KUKA KRL program: edge_4_right_mte.src, edge_4_right_mte.dat

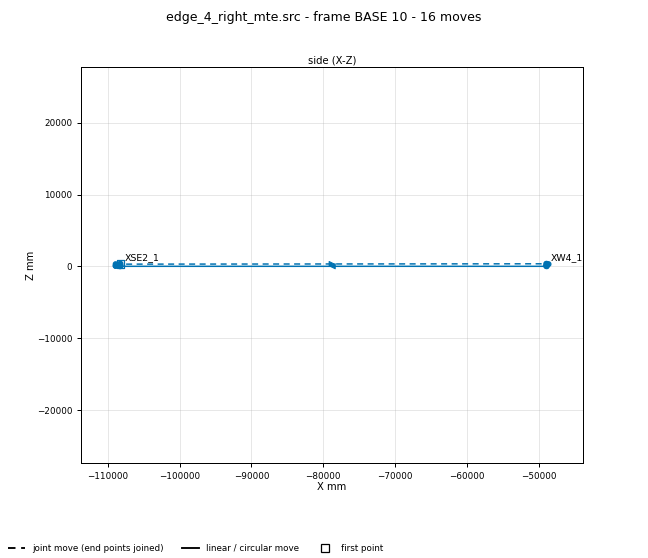
[picture p0: tool path of edge_4_right_mte.src in frame BASE 10, 16 of 16 moves have a stored position in this frame; points joined in program order, loops and branches not executed]
--- edge_4_right_mte.src ---
&ACCESS RVP
&REL 45
&PARAM EDITMASK = *
&PARAM DISKPATH = KRC:\R1\Program
DEF edge_4_right_mte( )
;FOLD INI;%{PE}
  ;FOLD BASISTECH INI
    GLOBAL INTERRUPT DECL 3 WHEN $STOPMESS==TRUE DO IR_STOPM ( )
    INTERRUPT ON 3
    BAS (#INITMOV,0 )
  ;ENDFOLD (BASISTECH INI)
  ;FOLD USER INI
    ;Make your modifications here

  ;ENDFOLD (USER INI)
;ENDFOLD (INI)
TS_CorrOff()
;FOLD PTP SE2_1 Vel= 100 % PDATW1_1 Tool[1] Base[10] ;%{PE}%R 8.3.34,%MKUKATPBASIS,%CMOVE,%VPTP,%P 1:PTP, 2:SE2_1, 3:C_DIS, 5:100, 7:PDATSE2_1
$BWDSTART = FALSE
PDAT_ACT=PPDATSE2_1
FDAT_ACT=FSE2_1
BAS(#PTP_PARAMS,100)
SET_CD_PARAMS (0)
PTP XSE2_1 C_DIS
;ENDFOLD

;FOLD LIN SE2_2 Vel= 0.06 m/s CPDATSE2_2 TouchSense SEARCH VIA SE2_3 CDSE2_2 SPSE2_2 Tool[1] Base[10] ;%{PE}
;FOLD Parameters ;%{h}
;Params IlfProvider=kukaroboter.touchsense.searchlin; Kuka.PointName=SE2_2; Kuka.BlendingEnabled=False; Kuka.MoveDataName=CPDATSE2_2; Kuka.VelocityPath=0.06; Kuka.MovementParameterFieldEnabled=True; MoveType=LIN
;FOLD Parameters TouchSense ;%{h}
;Params TouchSense.SearchViaPoint=SE2_3;TouchSense.ReferenceMove=CDSE2_2;TouchSense.SeachParam=SPSE2_2
;ENDFOLD
;ENDFOLD
$BWDSTART = FALSE
LDAT_ACT=LCPDATSE2_2
FDAT_ACT=FSE2_2
BAS(#CP_PARAMS,0.06)
SET_CD_PARAMS (0)
LIN XSE2_2 C_DIS C_DIS
TS_InitMovement($POS_ACT, XSE2_3, ZSPSE2_2)
TS_ManMoveToVia(XSE2_3)
TS_Search(XSE2_3, ZSPSE2_2, VCDSE2_2)
TS_SetCorrData(ZSPSE2_2, VCDSE2_2)
;ENDFOLD

;FOLD TouchSense Corr 1 CDSE2_2;%{E}
;FOLD Parameters Corr 1D ;%{h}
;Params IlfProvider=KukaRoboter.TouchSense.Correction1D;Correction1D=CDSE2_2
;ENDFOLD
TS_BC6DCalc(VCDSE2_2, TSg_CD0, TSg_CD0, TSg_CD0, TSg_CD0, TSg_CD0)
;ENDFOLD

;FOLD LIN SE2_4 Vel= 0.06 m/s CPDATSE2_4 TouchSense SEARCH VIA SE2_5 CDSE2_4 SPSE2_4 Tool[1] Base[10] ;%{PE}
;FOLD Parameters ;%{h}
;Params IlfProvider=kukaroboter.touchsense.searchlin; Kuka.PointName=SE2_4; Kuka.BlendingEnabled=False; Kuka.MoveDataName=CPDATSE2_4; Kuka.VelocityPath=0.06; Kuka.MovementParameterFieldEnabled=True; MoveType=LIN
;FOLD Parameters TouchSense ;%{h}
;Params TouchSense.SearchViaPoint=SE2_5;TouchSense.ReferenceMove=CDSE2_4;TouchSense.SeachParam=SPSE2_4
;ENDFOLD
;ENDFOLD
$BWDSTART = FALSE
LDAT_ACT=LCPDATSE2_4
FDAT_ACT=FSE2_4
BAS(#CP_PARAMS,0.06)
SET_CD_PARAMS (0)
LIN XSE2_4 C_DIS C_DIS
TS_InitMovement($POS_ACT, XSE2_5, ZSPSE2_4)
TS_ManMoveToVia(XSE2_5)
TS_Search(XSE2_5, ZSPSE2_4, VCDSE2_4)
TS_SetCorrData(ZSPSE2_4, VCDSE2_4)
;ENDFOLD

;FOLD TouchSense Corr 2 CDSE2_2 CDSE2_4;%{E}
;FOLD Parameters Corr 2D ;%{h}
;Params IlfProvider=KukaRoboter.TouchSense.Correction2D;Correction1D=CDSE2_2;Correction2D=CDSE2_4
;ENDFOLD
TS_BC6DCalc(VCDSE2_2, TSg_CD0, TSg_CD0, VCDSE2_4, TSg_CD0, TSg_CD0)
;ENDFOLD

;FOLD LIN SE2_6 Vel= 0.06 m/s CPDATS1_2 Tool[1] Base[10] ;%{PE}%R 8.3.34,%MKUKATPBASIS,%CMOVE,%VLIN,%P 1:LIN, 2:SE2_6, 3:, 5:0.06, 7:CPDATSE2_6
$BWDSTART = FALSE
LDAT_ACT=LCPDATSE2_6
FDAT_ACT=FSE2_6
BAS(#CP_PARAMS,0.06)
SET_CD_PARAMS (0)
LIN XSE2_6 C_DIS C_DIS
;ENDFOLD

;FOLD LIN SE2_7 Vel= 0.02 m/s CPDATSE2_7 TouchSense SEARCH VIA SE2_8 CDSE2_7 SPSE2_7 Tool[1] Base[10] ;%{PE}
;FOLD Parameters ;%{h}
;Params IlfProvider=kukaroboter.touchsense.searchlin; Kuka.PointName=SE2_7; Kuka.BlendingEnabled=False; Kuka.MoveDataName=CPDATSE2_7; Kuka.VelocityPath=0.02; Kuka.MovementParameterFieldEnabled=True; MoveType=LIN
;FOLD Parameters TouchSense ;%{h}
;Params TouchSense.SearchViaPoint=SE2_8;TouchSense.ReferenceMove=CDSE2_7;TouchSense.SeachParam=SPSE2_7
;ENDFOLD
;ENDFOLD
$BWDSTART = FALSE
LDAT_ACT=LCPDATSE2_7
FDAT_ACT=FSE2_7
BAS(#CP_PARAMS,0.02)
SET_CD_PARAMS (0)
LIN XSE2_7 C_DIS C_DIS
TS_InitMovement($POS_ACT, XSE2_8, ZSPSE2_7)
TS_ManMoveToVia(XSE2_8)
TS_Search(XSE2_8, ZSPSE2_7, VCDSE2_7)
TS_SetCorrData(ZSPSE2_7, VCDSE2_7)
;ENDFOLD

;FOLD TouchSense Corr 3 CDSE2_2 CDSE2_4 CDSE2_7;%{E}
;FOLD Parameters Corr 3D ;%{h}
;Params IlfProvider=KukaRoboter.TouchSense.Correction3D;Correction1D=CDSE2_2;Correction2D=CDSE2_4;Correction3D=CDSE2_7
;ENDFOLD
TS_BC6DCalc(VCDSE2_2, TSg_CD0, TSg_CD0, VCDSE2_4, TSg_CD0, VCDSE2_7)
;ENDFOLD

;FOLD LIN SE2_9 Vel= 0.1 m/s CPDATS1_2 Tool[1] Base[10] ;%{PE}%R 8.3.34,%MKUKATPBASIS,%CMOVE,%VLIN,%P 1:LIN, 2:SE2_9, 3:, 5:0.1, 7:CPDATSE2_9
$BWDSTART = FALSE
LDAT_ACT=LCPDATSE2_9
FDAT_ACT=FSE2_9
BAS(#CP_PARAMS,0.1)
SET_CD_PARAMS (0)
LIN XSE2_9 C_DIS C_DIS
;ENDFOLD

;FOLD PTP SS3_1 Vel= 100 % PDATW1_1 Tool[1] Base[10] ;%{PE}%R 8.3.34,%MKUKATPBASIS,%CMOVE,%VPTP,%P 1:PTP, 2:SS3_1, 3:C_DIS, 5:100, 7:PDATSS3_1
$BWDSTART = FALSE
PDAT_ACT=PPDATSS3_1
FDAT_ACT=FSS3_1
BAS(#PTP_PARAMS,100)
SET_CD_PARAMS (0)
PTP XSS3_1 C_DIS
;ENDFOLD

;FOLD LIN SS3_2 Vel= 0.06 m/s CPDATSS3_2 TouchSense SEARCH VIA SS3_3 CDSS3_2 SPSS3_2 Tool[1] Base[10] ;%{PE}
;FOLD Parameters ;%{h}
;Params IlfProvider=kukaroboter.touchsense.searchlin; Kuka.PointName=SS3_2; Kuka.BlendingEnabled=False; Kuka.MoveDataName=CPDATSS3_2; Kuka.VelocityPath=0.06; Kuka.MovementParameterFieldEnabled=True; MoveType=LIN
;FOLD Parameters TouchSense ;%{h}
;Params TouchSense.SearchViaPoint=SS3_3;TouchSense.ReferenceMove=CDSS3_2;TouchSense.SeachParam=SPSS3_2
;ENDFOLD
;ENDFOLD
$BWDSTART = FALSE
LDAT_ACT=LCPDATSS3_2
FDAT_ACT=FSS3_2
BAS(#CP_PARAMS,0.06)
SET_CD_PARAMS (0)
LIN XSS3_2 C_DIS C_DIS
TS_InitMovement($POS_ACT, XSS3_3, ZSPSS3_2)
TS_ManMoveToVia(XSS3_3)
TS_Search(XSS3_3, ZSPSS3_2, VCDSS3_2)
TS_SetCorrData(ZSPSS3_2, VCDSS3_2)
;ENDFOLD

;FOLD TouchSense Corr 1 CDSS3_2;%{E}
;FOLD Parameters Corr 1D ;%{h}
;Params IlfProvider=KukaRoboter.TouchSense.Correction1D;Correction1D=CDSS3_2
;ENDFOLD
TS_BC6DCalc(VCDSS3_2, TSg_CD0, TSg_CD0, TSg_CD0, TSg_CD0, TSg_CD0)
;ENDFOLD

;FOLD LIN SS3_4 Vel= 0.06 m/s CPDATSS3_4 TouchSense SEARCH VIA SS3_5 CDSS3_4 SPSS3_4 Tool[1] Base[10] ;%{PE}
;FOLD Parameters ;%{h}
;Params IlfProvider=kukaroboter.touchsense.searchlin; Kuka.PointName=SS3_4; Kuka.BlendingEnabled=False; Kuka.MoveDataName=CPDATSS3_4; Kuka.VelocityPath=0.06; Kuka.MovementParameterFieldEnabled=True; MoveType=LIN
;FOLD Parameters TouchSense ;%{h}
;Params TouchSense.SearchViaPoint=SS3_5;TouchSense.ReferenceMove=CDSS3_4;TouchSense.SeachParam=SPSS3_4
;ENDFOLD
;ENDFOLD
$BWDSTART = FALSE
LDAT_ACT=LCPDATSS3_4
FDAT_ACT=FSS3_4
BAS(#CP_PARAMS,0.06)
SET_CD_PARAMS (0)
LIN XSS3_4 C_DIS C_DIS
TS_InitMovement($POS_ACT, XSS3_5, ZSPSS3_4)
TS_ManMoveToVia(XSS3_5)
TS_Search(XSS3_5, ZSPSS3_4, VCDSS3_4)
TS_SetCorrData(ZSPSS3_4, VCDSS3_4)
;ENDFOLD

;FOLD TouchSense Corr 2 CDSS3_2 CDSS3_4;%{E}
;FOLD Parameters Corr 2D ;%{h}
;Params IlfProvider=KukaRoboter.TouchSense.Correction2D;Correction1D=CDSS3_2;Correction2D=CDSS3_4
;ENDFOLD
TS_BC6DCalc(VCDSS3_2, TSg_CD0, TSg_CD0, VCDSS3_4, TSg_CD0, TSg_CD0)
;ENDFOLD

;FOLD LIN SS3_6 Vel= 0.1 m/s CPDATS1_2 Tool[1] Base[10] ;%{PE}%R 8.3.34,%MKUKATPBASIS,%CMOVE,%VLIN,%P 1:LIN, 2:SS3_6, 3:, 5:0.1, 7:CPDATSS3_6
$BWDSTART = FALSE
LDAT_ACT=LCPDATSS3_6
FDAT_ACT=FSS3_6
BAS(#CP_PARAMS,0.1)
SET_CD_PARAMS (0)
LIN XSS3_6 C_DIS C_DIS
;ENDFOLD

;FOLD PTP W4_1 Vel= 100 % PDATW1_1 Tool[1] Base[10] ;%{PE}%R 8.3.34,%MKUKATPBASIS,%CMOVE,%VPTP,%P 1:PTP, 2:W4_1, 3:C_DIS, 5:100, 7:PDATW4_1
$BWDSTART = FALSE
PDAT_ACT=PPDATW4_1
FDAT_ACT=FW4_1
BAS(#PTP_PARAMS,100)
SET_CD_PARAMS (0)
PTP XW4_1 C_DIS
;ENDFOLD

;FOLD LIN W4_2 Vel= 0.2 m/s CPDATS1_2 Tool[1] Base[10] ;%{PE}%R 8.3.34,%MKUKATPBASIS,%CMOVE,%VLIN,%P 1:LIN, 2:W4_2, 3:, 5:0.2, 7:CPDATW4_2
$BWDSTART = FALSE
LDAT_ACT=LCPDATW4_2
FDAT_ACT=FW4_2
BAS(#CP_PARAMS,0.2)
SET_CD_PARAMS (0)
LIN XW4_2 C_DIS C_DIS
;ENDFOLD

custom_sync('hFAFA0000', 'hffff0000', 250)

;FOLD ARCON WDATW4_3 LIN W4_3 Vel= 0.1 m/s CPDATW8_4 Tool[1] Base[10];%{PE}
;FOLD Parameters ;%{h}
;Params IlfProvider=kukaroboter.arctech.arconlin; Kuka.PointName=W4_3; Kuka.BlendingEnabled=False; Kuka.MoveDataName=CPDATW4_3; Kuka.VelocityPath=0.1; Kuka.CurrentCDSetIndex=0; Kuka.MovementParameterFieldEnabled=True; ArcTech.WdatVarName=WDATW4_3
;ENDFOLD
$BWDSTART = FALSE
LDAT_ACT = LCPDATW4_3
FDAT_ACT = FW4_3
BAS(#CP_PARAMS,0.1)
SET_CD_PARAMS (0)
TRIGGER WHEN DISTANCE = 1 DELAY = ArcGetDelay(#PreDefinition, WDATW4_3) DO ArcMainNG(#PreDefinition, WDATW4_3, WW4_3) PRIO = -1
TRIGGER WHEN PATH = ArcGetPath(#OnTheFlyArcOn, WDATW4_3) DELAY = ArcGetDelay(#GasPreflow, WDATW4_3) DO ArcMainNG(#GasPreflow, WDATW4_3, WW4_3) PRIO = -1
TRIGGER WHEN PATH = ArcGetPath(#OnTheFlyArcOn, WDATW4_3) DELAY = 0 DO ArcMainNG(#ArcOnMoveStd, WDATW4_3, WW4_3) PRIO = -1
ArcMainNG(#ArcOnBeforeMoveStd, WDATW4_3, WW4_3)
LIN XW4_3
ArcMainNG(#ArcOnAfterMoveStd, WDATW4_3, WW4_3)
;ENDFOLD

;FOLD ARCOFF WDATW4_4 LIN W4_4 CPDATW4_4 Tool[1] Base[10];%{PE}
;FOLD Parameters ;%{h}
;Params IlfProvider=kukaroboter.arctech.arcofflin; Kuka.IsGlobalPoint=False; Kuka.PointName=W4_4; Kuka.BlendingEnabled=False; Kuka.MoveDataName=CPDATW4_4; Kuka.VelocityPath=0.0063; Kuka.CurrentCDSetIndex=0; Kuka.MovementParameterFieldEnabled=True; ArcTech.WdatVarName=WDATW4_4
;ENDFOLD
$BWDSTART = FALSE
LDAT_ACT = LCPDATW4_4
FDAT_ACT = FW4_4
BAS(#CP_PARAMS, gArcBasVelDefinition)
SET_CD_PARAMS (0)
TRIGGER WHEN PATH = ArcGetPath(#ArcOffBefore, WDATW4_4) DELAY = 0 DO ArcMainNG(#ArcOffBeforeOffStd, WDATW4_4) PRIO = -1
TRIGGER WHEN PATH = ArcGetPath(#OnTheFlyArcOff, WDATW4_4) DELAY = 0 DO ArcMainNG(#ArcOffMoveStd, WDATW4_4) PRIO = -1
ArcMainNG(#ArcOffBeforeMoveStd, WDATW4_4)
LIN XW4_4
ArcMainNG(#ArcOffAfterMoveStd, WDATW4_4)
;ENDFOLD

;FOLD LIN W4_5 Vel= 0.2 m/s CPDATS1_2 Tool[1] Base[10] ;%{PE}%R 8.3.34,%MKUKATPBASIS,%CMOVE,%VLIN,%P 1:LIN, 2:W4_5, 3:, 5:0.2, 7:CPDATW4_5
$BWDSTART = FALSE
LDAT_ACT=LCPDATW4_5
FDAT_ACT=FW4_5
BAS(#CP_PARAMS,0.2)
SET_CD_PARAMS (0)
LIN XW4_5 C_DIS C_DIS
;ENDFOLD

;FOLD LIN W4_6 Vel= 0.4 m/s CPDATS1_2 Tool[1] Base[10] ;%{PE}%R 8.3.34,%MKUKATPBASIS,%CMOVE,%VLIN,%P 1:LIN, 2:W4_6, 3:, 5:0.4, 7:CPDATW4_6
$BWDSTART = FALSE
LDAT_ACT=LCPDATW4_6
FDAT_ACT=FW4_6
BAS(#CP_PARAMS,0.4)
SET_CD_PARAMS (0)
LIN XW4_6 C_DIS C_DIS
;ENDFOLD

TS_CorrOff()
ochistka_mod()
END

--- edge_4_right_mte.dat ---
&ACCESS RVP
&REL 45
&PARAM EDITMASK = *
&PARAM DISKPATH = KRC:\R1\Program
DEFDAT  edge_4_right_mte
;FOLD EXTERNAL DECLARATIONS;%{PE}%MKUKATPBASIS,%CEXT,%VCOMMON,%P
;FOLD BASISTECH EXT;%{PE}%MKUKATPBASIS,%CEXT,%VEXT,%P
EXT  BAS (BAS_COMMAND  :IN,REAL  :IN )
DECL INT SUCCESS
;ENDFOLD (BASISTECH EXT)
;FOLD USER EXT;%{E}%MKUKATPUSER,%CEXT,%VEXT,%P
;Make your modifications here

;ENDFOLD (USER EXT)
;ENDFOLD (EXTERNAL DECLARATIONS)

DECL PDAT PPDATSE2_1={VEL 100,ACC 100.0,APO_DIST 10.0,GEAR_JERK 50.0000,EXAX_IGN 0}
DECL FDAT FSE2_1={TOOL_NO 1,BASE_NO 10,IPO_FRAME #BASE,POINT2[] " "}
DECL E6POS XSE2_1={X -108215.0,Y 2768.0,Z 366.0,A -45,B 50,C -180,S 20,T 53,E1 -10000,E2 0,E3 1800,E4 0,E5 0,E6 0}

DECL E6POS XSE2_2={X -108215.0,Y 2768.0,Z 76.0,A -45,B 50,C -180,S 20,T 53,E1 -10000,E2 0,E3 1800,E4 0,E5 0,E6 0}
DECL FDAT FSE2_2={TOOL_NO 1,BASE_NO 10,IPO_FRAME #BASE,POINT2[] " ",TQ_STATE FALSE}
DECL LDAT LCPDATSE2_2={VEL 0.06,ACC 100.0,APO_DIST 10.0,APO_FAC 50.0,ORI_TYP #VAR,CIRC_TYP #BASE,JERK_FAC 50.0}
DECL E6POS XSE2_3={X -108215.0,Y 2768.0,Z 16.0,A -45,B 50,C -180,S 20,T 53,E1 -10000,E2 0,E3 1800,E4 0,E5 0,E6 0}
DECL FDAT FSE2_3={TOOL_NO 1,BASE_NO 10,IPO_FRAME #BASE,POINT2[] " ",TQ_STATE FALSE}
DECL TSg_PCollCD_T VCDSE2_2={CD_IPO_MODE #BASE,Mastered TRUE,SDir_W {X 0.0,Y 0.0,Z 0.0,A 0.0,B 0.0,C 0.0},Ref_W {X -108215.0,Y 2768.0,Z 16.0,A -45,B 50,C -180},Meas_W {X 0.0,Y 0.0,Z 0.0,A 0.0,B 0.0,C 0.0},Diff_W {X 0.0,Y 0.0,Z 0.0,A 0.0,B 0.0,C 0.0},VecLenDiff_W 0.0,MEnum #CDEmpty,MC 1}
DECL TSg_SearchProperty_T ZSPSE2_2={MoveType #MoveWithLin,TouchType #Single,DynamicStep #Slow,SensorNum 1,SearchDepth_Tol 150.0,bBackToStartPos TRUE}

DECL E6POS XSE2_4={X -108215.0,Y 2768.0,Z 76.0,A -60,B 50,C 169,S 20,T 53,E1 -10000,E2 0,E3 1800,E4 0,E5 0,E6 0}
DECL FDAT FSE2_4={TOOL_NO 1,BASE_NO 10,IPO_FRAME #BASE,POINT2[] " ",TQ_STATE FALSE}
DECL LDAT LCPDATSE2_4={VEL 0.06,ACC 100.0,APO_DIST 10.0,APO_FAC 50.0,ORI_TYP #VAR,CIRC_TYP #BASE,JERK_FAC 50.0}
DECL E6POS XSE2_5={X -108215.0,Y 2708.0,Z 76.0,A -60,B 50,C 169,S 20,T 53,E1 -10000,E2 0,E3 1800,E4 0,E5 0,E6 0}
DECL FDAT FSE2_5={TOOL_NO 1,BASE_NO 10,IPO_FRAME #BASE,POINT2[] " ",TQ_STATE FALSE}
DECL TSg_PCollCD_T VCDSE2_4={CD_IPO_MODE #BASE,Mastered TRUE,SDir_W {X 0.0,Y 0.0,Z 0.0,A 0.0,B 0.0,C 0.0},Ref_W {X -108215.0,Y 2708.0,Z 76.0,A -60,B 50,C 169},Meas_W {X 0.0,Y 0.0,Z 0.0,A 0.0,B 0.0,C 0.0},Diff_W {X 0.0,Y 0.0,Z 0.0,A 0.0,B 0.0,C 0.0},VecLenDiff_W 0.0,MEnum #CDEmpty,MC 1}
DECL TSg_SearchProperty_T ZSPSE2_4={MoveType #MoveWithLin,TouchType #Single,DynamicStep #Slow,SensorNum 1,SearchDepth_Tol 150.0,bBackToStartPos TRUE}

DECL LDAT LCPDATSE2_6={VEL 0.06,ACC 100.0,APO_DIST 10.0,APO_FAC 50.0,ORI_TYP #VAR,CIRC_TYP #BASE,JERK_FAC 50.0,GEAR_JERK 50.0000,EXAX_IGN 0}
DECL FDAT FSE2_6={TOOL_NO 1,BASE_NO 10,IPO_FRAME #BASE,POINT2[] " "}
DECL E6POS XSE2_6={X -108890.0,Y 2768.0,Z 76.0,A -30,B 40,C -169,S 20,T 53,E1 -10000,E2 0,E3 1800,E4 0,E5 0,E6 0}

DECL E6POS XSE2_7={X -108890.0,Y 2698.0,Z 76.0,A -30,B 40,C -169,S 20,T 53,E1 -10000,E2 0,E3 1800,E4 0,E5 0,E6 0}
DECL FDAT FSE2_7={TOOL_NO 1,BASE_NO 10,IPO_FRAME #BASE,POINT2[] " ",TQ_STATE FALSE}
DECL LDAT LCPDATSE2_7={VEL 0.02,ACC 100.0,APO_DIST 10.0,APO_FAC 50.0,ORI_TYP #VAR,CIRC_TYP #BASE,JERK_FAC 50.0}
DECL E6POS XSE2_8={X -108830.0,Y 2698.0,Z 76.0,A -30,B 40,C -169,S 20,T 53,E1 -10000,E2 0,E3 1800,E4 0,E5 0,E6 0}
DECL FDAT FSE2_8={TOOL_NO 1,BASE_NO 10,IPO_FRAME #BASE,POINT2[] " ",TQ_STATE FALSE}
DECL TSg_PCollCD_T VCDSE2_7={CD_IPO_MODE #BASE,Mastered TRUE,SDir_W {X 0.0,Y 0.0,Z 0.0,A 0.0,B 0.0,C 0.0},Ref_W {X -108830.0,Y 2698.0,Z 76.0,A -30,B 40,C -169},Meas_W {X 0.0,Y 0.0,Z 0.0,A 0.0,B 0.0,C 0.0},Diff_W {X 0.0,Y 0.0,Z 0.0,A 0.0,B 0.0,C 0.0},VecLenDiff_W 0.0,MEnum #CDEmpty,MC 1}
DECL TSg_SearchProperty_T ZSPSE2_7={MoveType #MoveWithLin,TouchType #Single,DynamicStep #Slow,SensorNum 1,SearchDepth_Tol 150.0,bBackToStartPos TRUE}

DECL LDAT LCPDATSE2_9={VEL 0.1,ACC 100.0,APO_DIST 10.0,APO_FAC 50.0,ORI_TYP #VAR,CIRC_TYP #BASE,JERK_FAC 50.0,GEAR_JERK 50.0000,EXAX_IGN 0}
DECL FDAT FSE2_9={TOOL_NO 1,BASE_NO 10,IPO_FRAME #BASE,POINT2[] " "}
DECL E6POS XSE2_9={X -108890.0,Y 2768.0,Z 316.0,A -30,B 50,C -169,S 20,T 53,E1 -10000,E2 0,E3 1800,E4 0,E5 0,E6 0}

DECL PDAT PPDATSS3_1={VEL 100,ACC 100.0,APO_DIST 10.0,GEAR_JERK 50.0000,EXAX_IGN 0}
DECL FDAT FSS3_1={TOOL_NO 1,BASE_NO 10,IPO_FRAME #BASE,POINT2[] " "}
DECL E6POS XSS3_1={X -48957.5,Y 2768.0,Z 366.0,A -120,B 50,C -180,S 20,T 53,E1 -10000,E2 0,E3 1800,E4 0,E5 0,E6 0}

DECL E6POS XSS3_2={X -48957.5,Y 2768.0,Z 76.0,A -120,B 50,C -180,S 20,T 53,E1 -10000,E2 0,E3 1800,E4 0,E5 0,E6 0}
DECL FDAT FSS3_2={TOOL_NO 1,BASE_NO 10,IPO_FRAME #BASE,POINT2[] " ",TQ_STATE FALSE}
DECL LDAT LCPDATSS3_2={VEL 0.06,ACC 100.0,APO_DIST 10.0,APO_FAC 50.0,ORI_TYP #VAR,CIRC_TYP #BASE,JERK_FAC 50.0}
DECL E6POS XSS3_3={X -48957.5,Y 2768.0,Z 16.0,A -120,B 50,C -180,S 20,T 53,E1 -10000,E2 0,E3 1800,E4 0,E5 0,E6 0}
DECL FDAT FSS3_3={TOOL_NO 1,BASE_NO 10,IPO_FRAME #BASE,POINT2[] " ",TQ_STATE FALSE}
DECL TSg_PCollCD_T VCDSS3_2={CD_IPO_MODE #BASE,Mastered TRUE,SDir_W {X 0.0,Y 0.0,Z 0.0,A 0.0,B 0.0,C 0.0},Ref_W {X -48957.5,Y 2768.0,Z 16.0,A -120,B 50,C -180},Meas_W {X 0.0,Y 0.0,Z 0.0,A 0.0,B 0.0,C 0.0},Diff_W {X 0.0,Y 0.0,Z 0.0,A 0.0,B 0.0,C 0.0},VecLenDiff_W 0.0,MEnum #CDEmpty,MC 1}
DECL TSg_SearchProperty_T ZSPSS3_2={MoveType #MoveWithLin,TouchType #Single,DynamicStep #Slow,SensorNum 1,SearchDepth_Tol 150.0,bBackToStartPos TRUE}

DECL E6POS XSS3_4={X -48957.5,Y 2768.0,Z 76.0,A -120,B 50,C 169,S 20,T 53,E1 -10000,E2 0,E3 1800,E4 0,E5 0,E6 0}
DECL FDAT FSS3_4={TOOL_NO 1,BASE_NO 10,IPO_FRAME #BASE,POINT2[] " ",TQ_STATE FALSE}
DECL LDAT LCPDATSS3_4={VEL 0.06,ACC 100.0,APO_DIST 10.0,APO_FAC 50.0,ORI_TYP #VAR,CIRC_TYP #BASE,JERK_FAC 50.0}
DECL E6POS XSS3_5={X -48957.5,Y 2708.0,Z 76.0,A -120,B 50,C 169,S 20,T 53,E1 -10000,E2 0,E3 1800,E4 0,E5 0,E6 0}
DECL FDAT FSS3_5={TOOL_NO 1,BASE_NO 10,IPO_FRAME #BASE,POINT2[] " ",TQ_STATE FALSE}
DECL TSg_PCollCD_T VCDSS3_4={CD_IPO_MODE #BASE,Mastered TRUE,SDir_W {X 0.0,Y 0.0,Z 0.0,A 0.0,B 0.0,C 0.0},Ref_W {X -48957.5,Y 2708.0,Z 76.0,A -120,B 50,C 169},Meas_W {X 0.0,Y 0.0,Z 0.0,A 0.0,B 0.0,C 0.0},Diff_W {X 0.0,Y 0.0,Z 0.0,A 0.0,B 0.0,C 0.0},VecLenDiff_W 0.0,MEnum #CDEmpty,MC 1}
DECL TSg_SearchProperty_T ZSPSS3_4={MoveType #MoveWithLin,TouchType #Single,DynamicStep #Slow,SensorNum 1,SearchDepth_Tol 150.0,bBackToStartPos TRUE}

DECL LDAT LCPDATSS3_6={VEL 0.1,ACC 100.0,APO_DIST 10.0,APO_FAC 50.0,ORI_TYP #VAR,CIRC_TYP #BASE,JERK_FAC 50.0,GEAR_JERK 50.0000,EXAX_IGN 0}
DECL FDAT FSS3_6={TOOL_NO 1,BASE_NO 10,IPO_FRAME #BASE,POINT2[] " "}
DECL E6POS XSS3_6={X -48637.5,Y 2768.0,Z 316.0,A -150,B 50,C -169,S 20,T 53,E1 -10000,E2 0,E3 1800,E4 0,E5 0,E6 0}

DECL PDAT PPDATW4_1={VEL 100,ACC 100.0,APO_DIST 10.0,GEAR_JERK 50.0000,EXAX_IGN 0}
DECL FDAT FW4_1={TOOL_NO 1,BASE_NO 10,IPO_FRAME #BASE,POINT2[] " "}
DECL E6POS XW4_1={X -48897.5,Y 2768.0,Z 366.0,A -118.5,B 41.3,C 160.3,S 20,T 53,E1 -10000,E2 0,E3 1800,E4 0,E5 0,E6 0}

DECL LDAT LCPDATW4_2={VEL 0.2,ACC 100.0,APO_DIST 10.0,APO_FAC 50.0,ORI_TYP #VAR,CIRC_TYP #BASE,JERK_FAC 50.0,GEAR_JERK 50.0000,EXAX_IGN 0}
DECL FDAT FW4_2={TOOL_NO 1,BASE_NO 10,IPO_FRAME #BASE,POINT2[] " "}
DECL E6POS XW4_2={X -48897.5,Y 2768.0,Z 76.0,A -118.5,B 41.3,C 160.3,S 20,T 53,E1 -10000,E2 0,E3 1800,E4 0,E5 0,E6 0}

DECL stArcDat_T WDATW4_3={Strike {JobModeId[] "Job Mode",ParamSetId[] "Set1",StartTime 0.0,PreFlowTime 0.0,Channel1 1,Channel2 0.0,Channel3 0.0,Channel4 0.0,Channel5 0.0,Channel6 0.0,Channel7 0.0,Channel8 0.0,PurgeTime 0.0},Weld {JobModeId[] "Job Mode",ParamSetId[] "Set2",Velocity 0.0063,Channel1 1,Channel2 0,Channel3 0.0,Channel4 0.0,Channel5 0.0,Channel6 0.0,Channel7 0.0,Channel8 0.0},Weave {Pattern #Triangle,Length 3.5,Amplitude 2,Angle 0.0,LeftSideDelay 0.0,RightSideDelay 0.0},Advanced {IgnitionErrorStrategy 1,WeldErrorStrategy 1,SlopeOption #None,SlopeTime 0.0,SlopeDistance 0.0,OnTheFlyActiveOn FALSE,OnTheFlyActiveOff FALSE,OnTheFlyDistanceOn 0.0,OnTheFlyDistanceOff 0.0},Track {IsArcSenseEnabled TRUE,ControlEnabled TRUE,KeepOffset TRUE,TeachNew FALSE,FindSeamMiddle TRUE,TrackingDelay 0.2,ControlSensibility 25.0,MaxDeviation 100,ControlSensibilityHeight 25.0,Bias 0.0,WeaveOffset 0.0,HeightCorrValue 0.0}}
DECL stArcDat_T WW4_3={Strike {SeamName[] " ",SeamNumber -1},Advanced {BitCodedRobotMark 0}}
DECL E6POS XW4_3={X -48897.5,Y 2708.0,Z 16.0,A -118.5,B 41.3,C 160.3,S 20,T 53,E1 -10000,E2 0,E3 1800,E4 0,E5 0,E6 0}
DECL FDAT FW4_3={TOOL_NO 1,BASE_NO 10,IPO_FRAME #BASE,POINT2[] " "}
DECL LDAT LCPDATW4_3={VEL 0.1,ACC 100.0,APO_DIST 0.0,APO_FAC 50.0,AXIS_VEL 100.0,AXIS_ACC 100.0,ORI_TYP #VAR,CIRC_TYP #BASE,JERK_FAC 50.0,GEAR_JERK 50.0,EXAX_IGN 0}

DECL stArcDat_T WDATW4_4={Crater {JobModeId[] "Job Mode",ParamSetId[] "Set3",CraterTime 0.0,PostflowTime 0.0,Channel1 1,Channel2 0.0,Channel3 0.0,Channel4 0.0,Channel5 0.0,Channel6 0.0,Channel7 0.0,Channel8 0.0,BurnBackTime 0.0},Advanced {IgnitionErrorStrategy 1,WeldErrorStrategy 1,SlopeOption #None,SlopeTime 0.0,SlopeDistance 0.0,OnTheFlyActiveOn FALSE,OnTheFlyActiveOff FALSE,OnTheFlyDistanceOn 0.0,OnTheFlyDistanceOff 0.0}}
DECL E6POS XW4_4={X -108273.0,Y 2708.0,Z 15.0,A -118.5,B 41.3,C 160.3,S 20,T 53,E1 -10000,E2 0,E3 1800,E4 0,E5 0,E6 0}
DECL FDAT FW4_4={TOOL_NO 1,BASE_NO 10,IPO_FRAME #BASE,POINT2[] " "}
DECL LDAT LCPDATW4_4={VEL 0.01,ACC 100.0,APO_DIST 0.0,APO_FAC 50.0,AXIS_VEL 100.0,AXIS_ACC 100.0,ORI_TYP #VAR,CIRC_TYP #BASE,JERK_FAC 50.0,GEAR_JERK 50.0,EXAX_IGN 0}

DECL LDAT LCPDATW4_5={VEL 0.2,ACC 100.0,APO_DIST 10.0,APO_FAC 50.0,ORI_TYP #VAR,CIRC_TYP #BASE,JERK_FAC 50.0,GEAR_JERK 50.0000,EXAX_IGN 0}
DECL FDAT FW4_5={TOOL_NO 1,BASE_NO 10,IPO_FRAME #BASE,POINT2[] " "}
DECL E6POS XW4_5={X -108273.0,Y 2768.0,Z 75.0,A -118.5,B 41.3,C 160.3,S 20,T 53,E1 -10000,E2 0,E3 1800,E4 0,E5 0,E6 0}

DECL LDAT LCPDATW4_6={VEL 0.4,ACC 100.0,APO_DIST 10.0,APO_FAC 50.0,ORI_TYP #VAR,CIRC_TYP #BASE,JERK_FAC 50.0,GEAR_JERK 50.0000,EXAX_IGN 0}
DECL FDAT FW4_6={TOOL_NO 1,BASE_NO 10,IPO_FRAME #BASE,POINT2[] " "}
DECL E6POS XW4_6={X -108273.0,Y 2768.0,Z 365.0,A -118.5,B 41.3,C 160.3,S 20,T 53,E1 -10000,E2 0,E3 1800,E4 0,E5 0,E6 0}
ENDDAT
